FUNCTION_BLOCK FB_FT_PI (* Composite Function Block Type *)
  (* Standard: 61499-2 *)
  (* Version 0.0, 2011-07-15, 4DIAC-IDE, 4DIAC-Consortium *)
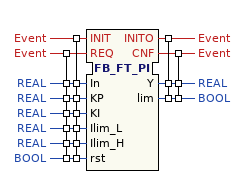
  EVENT_INPUT
    INIT WITH In, KP, KI, Ilim_L, Ilim_H, rst; (* Initialization Request *)
    REQ WITH In, KP, KI, Ilim_L, Ilim_H, rst; (* Normal Execution Request *)
  END_EVENT
  EVENT_OUTPUT
    INITO WITH Y, lim; (* Initialization Confirm *)
    CNF WITH Y, lim; (* Execution Confirmation *)
  END_EVENT
  VAR_INPUT
    In : REAL; (* Input value *)
    KP : REAL := 1.0; (* Amplification factor for proportional controller *)
    KI : REAL := 1.0; (* Amplification factor for integrator *)
    Ilim_L : REAL := -1E38; (* Minimal output value *)
    Ilim_H : REAL := 1E38; (* Maximal output value *)
    rst : BOOL; (* Reset output *)
  END_VAR
  VAR_OUTPUT
    Y : REAL; (* Output value *)
    lim : BOOL; (* Returns true if the limit is exceeded *)
  END_VAR
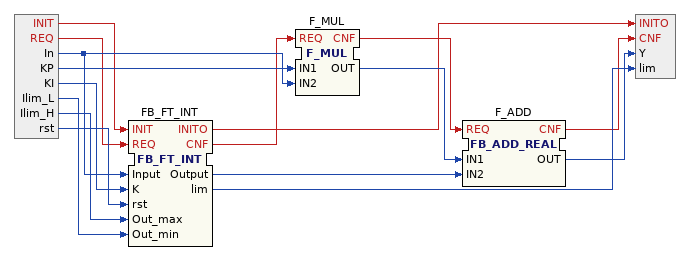
  FBS
    FB_FT_INT : FB_FT_INT;
    F_ADD : FB_ADD_REAL;
    F_MUL : F_MUL;
  END_FBS
  EVENT_CONNECTIONS
    INIT TO FB_FT_INT.INIT;
    FB_FT_INT.INITO TO INITO;
    REQ TO FB_FT_INT.REQ;
    FB_FT_INT.CNF TO F_MUL.REQ;
    F_MUL.CNF TO F_ADD.REQ;
    F_ADD.CNF TO CNF;
  END_CONNECTIONS
  DATA_CONNECTIONS
    In TO FB_FT_INT.Input;
    KI TO FB_FT_INT.K;
    rst TO FB_FT_INT.rst;
    Ilim_L TO FB_FT_INT.Out_min;
    Ilim_H TO FB_FT_INT.Out_max;
    FB_FT_INT.lim TO lim;
    KP TO F_MUL.IN1;
    In TO F_MUL.IN2;
    F_MUL.OUT TO F_ADD.IN1;
    FB_FT_INT.Output TO F_ADD.IN2;
    F_ADD.OUT TO Y;
  END_CONNECTIONS
END_FUNCTION_BLOCK
